TYPE ST_STATION_LIST_RESULT :
STRUCT
  wState    : WORD;   // wState == 0 --> all ok
  nIndex    : ULINT;
  stData    : ST_STATION_MOVER_DATA;  // copy of list entry
END_STRUCT
END_TYPE

(* stored: Version 1.1.0.1
   DUT ST_STATION_LIST_RESULT: Id {2fa78fdd-be8f-4df8-b727-a3b4446e3809} *)
